Fanuc KAREL source: kf00082.KL

-- PROVISIONAL review KL for V940-1; original PC SHA256 1e6b2a53a282748ed807f1654cf6b47d1fdf6c0529c005942869082c4037d8f8
-- Incomplete behavior may be omitted. Consult companion uncertainty JSON. Do not deploy.
PROGRAM KF00082
%NOLOCKGROUP
BEGIN
  -- V9_ZERO_TABLE_METADATA_HINT layout=0002_ascii; no indexed target words; source/name/runtime held
  -- UNRESOLVED_PC offsets 5-15; opcodes 27,22,31
  -- UNRESOLVED_PC offsets 20-54; opcodes 27,27,2E,22,22,22,22,31
  -- UNRESOLVED_PC offsets 59-93; opcodes 27,22,22,22,22,22,31
  -- UNRESOLVED_PC offsets 98-102; opcodes 7F
END KF00082
